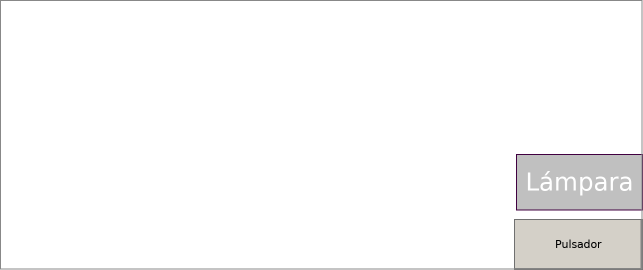
VISUALIZATION Visualization  // 643x270
    Rectangle (516,154 127x56), "Lámpara", colour toggle: MAIN.Lampara
    Button (514,219 129x51), "Pulsador"
        tap MAIN.Pulsador
END_VISUALIZATION

(* stored: Version 1.1.0.1, ProductVersion 3.1.4024.12
   Visu Visualization: Id {1e9fe31b-9e50-4ad6-8d77-4a8d4c6d6bf2} *)
